FUNCTION DWORD_TO_BYTE_ARRAY
VAR_INPUT
	Value	: DWORD;
END_VAR
VAR_IN_OUT
	DATA	: ARRAY [*] OF BYTE;
END_VAR
VAR
	i		: BYTE := 0;
END_VAR

FOR i := 0 TO 3 DO
	DATA[i] := DWORD_TO_BYTE(SHR(Value, (8*i)));			
END_FOR;

END_FUNCTION

(* stored: Version 1.1.0.1, ProductVersion 3.1.4024.11
   POU DWORD_TO_BYTE_ARRAY: Id {b245e009-a893-41c5-9455-bbd9fe187153}, SpecialFunc None *)
